(* IEC 61131-3 sources: axsharp/src/sanbox/integration/ix-integration-plc/SystemConstants, 2 files *)

(* ---- plc_line_HwIdentifiers.st ---- *)
CONFIGURATION HardwareIDs
    VAR_GLOBAL CONSTANT
        plc_line_HwID : UINT := UINT#32;
        plc_line_Rail_0_HwID : UINT := UINT#257;
        plc_line_plc_line_HwID : UINT := UINT#48;
        plc_line_plc_line_CPU_display_1_HwID : UINT := UINT#54;
        plc_line_plc_line_Card_reader_writer_1_HwID : UINT := UINT#51;
        plc_line_plc_line_OPC_UA_1_HwID : UINT := UINT#117;
        plc_line_plc_line_PROFINET_interface_1_HwID : UINT := UINT#64;
        plc_line_plc_line_PROFINET_interface_1_Port_1_HwID : UINT := UINT#65;
        plc_line_plc_line_PROFINET_interface_1_Port_2_HwID : UINT := UINT#66;
        plc_line_plc_line_PROFINET_interface_2_HwID : UINT := UINT#72;
        plc_line_plc_line_PROFINET_interface_2_Port_3_HwID : UINT := UINT#73;
        plc_line_plc_line_PROFINET_interface_2_Port_4_HwID : UINT := UINT#74;
        plc_line_plc_line_PROFINET_interface_GBIT_3_HwID : UINT := UINT#120;
        plc_line_plc_line_PROFINET_interface_GBIT_3_Port_5_HwID : UINT := UINT#121;
        plc_line_plc_line_Virtual_communication_interface_HwID : UINT := UINT#135;
        profinet_plc_line_HwID : UINT := UINT#256;

    END_VAR
END_CONFIGURATION

(* ---- plc_line_IoAddresses.st ---- *)
CONFIGURATION IoAddresses
    VAR_GLOBAL
    END_VAR
END_CONFIGURATION
